(* IEC 61131-3 sources: Py_iec/tests/fixtures/st/valid, 1 file *)

(* ---- counter.st ---- *)
FUNCTION_BLOCK Counter
VAR
    count : INT := 0;
END_VAR
count := count + 1;
END_FUNCTION_BLOCK
